PROGRAM Automatic
VAR
END_VAR

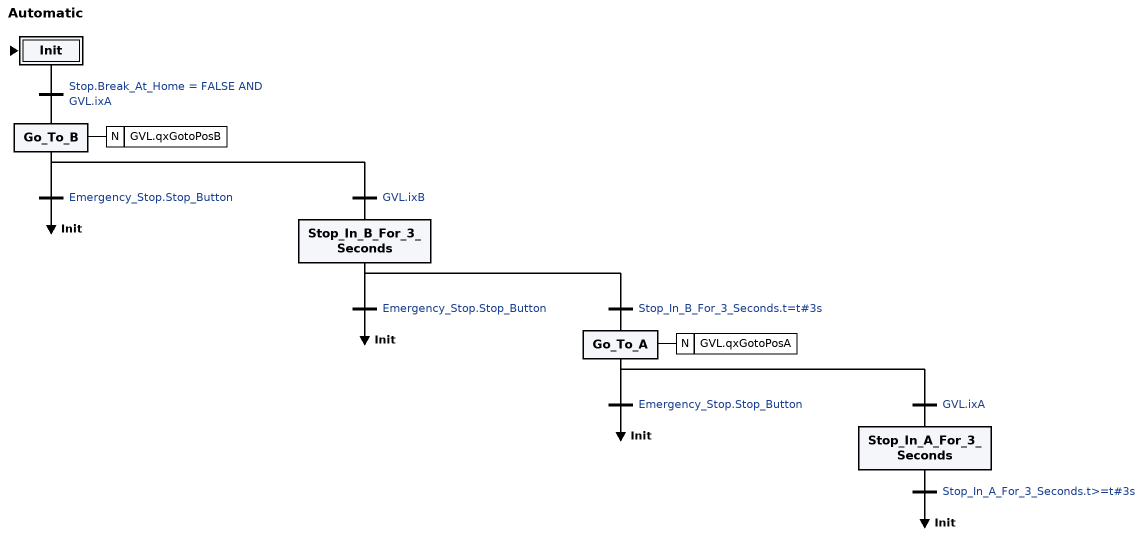
INITIAL_STEP Init:
END_STEP
TRANSITION FROM Init TO Go_To_B
    := Stop.Break_At_Home = FALSE AND GVL.ixA;
END_TRANSITION
STEP Go_To_B:
    GVL.qxGotoPosB(N);
END_STEP
TRANSITION FROM Go_To_B TO Init
    := Emergency_Stop.Stop_Button;
END_TRANSITION
TRANSITION FROM Go_To_B TO Stop_In_B_For_3_Seconds
    := GVL.ixB;
END_TRANSITION
STEP Stop_In_B_For_3_Seconds:
END_STEP
TRANSITION FROM Stop_In_B_For_3_Seconds TO Init
    := Emergency_Stop.Stop_Button;
END_TRANSITION
TRANSITION FROM Stop_In_B_For_3_Seconds TO Go_To_A
    := Stop_In_B_For_3_Seconds.t=t#3s;
END_TRANSITION
STEP Go_To_A:
    GVL.qxGotoPosA(N);
END_STEP
TRANSITION FROM Go_To_A TO Init
    := Emergency_Stop.Stop_Button;
END_TRANSITION
TRANSITION FROM Go_To_A TO Stop_In_A_For_3_Seconds
    := GVL.ixA;
END_TRANSITION
STEP Stop_In_A_For_3_Seconds:
END_STEP
TRANSITION FROM Stop_In_A_For_3_Seconds TO Init
    := Stop_In_A_For_3_Seconds.t>=t#3s;
END_TRANSITION

END_PROGRAM

(* stored: Version 1.1.0.1, ProductVersion 3.1.4024.12
   POU Automatic: Id {53b871c8-da1c-4d56-938d-022da038065b}, SpecialFunc None *)
